PROGRAM MAIN
VAR
END_VAR

END_PROGRAM

(* stored: Version 1.1.0.1
   POU MAIN: Id {ba5f6b21-102a-408e-8534-a49f454d6265} *)
